{attribute 'qualified_only'}
VAR_GLOBAL
	

  rX 			: REAL;
  rY			: REAL;
  iA			: INT;
  
  //mootor controls 
  
  bmotorstartpb 	: BOOL;
  bmotorstoppb		: BOOL;
  bmotorcontrol		: BOOL;
  
  bmotorcontrolenable : BOOL;
  
  
END_VAR

(* stored: Version 1.1.0.1, ProductVersion 3.1.4024.12
   GVL GVL: Id {d5471a99-fba4-4fb3-8f96-43c21058f870} *)
